PROGRAM POU
VAR
END_VAR

// NETWORK 1

END_PROGRAM

(* stored: Version 1.1.0.1, ProductVersion 3.1.4024.13
   POU POU: Id {6bf18b50-af56-416f-8587-1bd64ebd13fb}, SpecialFunc None *)
